(* LS Electric XG5000 project: plc_project_3 *)
(* PLC LSPLC *)

PROGRAM plc_storage (* task: 스캔 프로그램 *)
VAR
    CD : BOOL;
    CV : INT;
    ET : TIME;
    IN1 : BOOL;
    INST : TP;
    INST1 : TON;
    INST10 : TP;
    INST11 : TP;
    INST12 : TP;
    INST13 : TP;
    INST14 : TP;
    INST15 : TP;
    INST16 : TP;
    INST17 : TP;
    INST18 : TP;
    INST19 : TP;
    INST2 : TP;
    INST20 : TP;
    INST21 : TP;
    INST22 : TP;
    INST23 : TP;
    INST24 : TP;
    INST25 : TP;
    INST26 : TP;
    INST27 : TP;
    INST28 : TP;
    INST29 : TP;
    INST3 : TP;
    INST30 : TP;
    INST31 : TP;
    INST32 : TP;
    INST33 : TP;
    INST34 : TP;
    INST35 : TP;
    INST36 : TP;
    INST37 : TP;
    INST4 : TP;
    INST5 : TP;
    INST6 : TP;
    INST7 : TP;
    INST8 : TP;
    INST9 : TP;
    LD : BOOL;
    output1 : INT;
    output2 : UDINT;
    output3 : INT;
    output4 : UDINT;
    output5 : INT;
    output6 : UDINT;
    output7 : INT;
    output8 : UDINT;
    PV : INT;
    QD : BOOL;
    QU : BOOL;
    R : BOOL;
    time1 : TIME;
    time2 : TIME;
    time3 : TIME;
    time4 : TIME;
    난수1 : TON;
    난수2 : TON;
    난수3 : TON;
    놓기 AT %QX0.0.49 : BOOL;
    랜덤수 : INT;
    랜덤수2 : INT;
    반시계 AT %QX0.0.62 : BOOL;
    상 AT %QX0.0.60 : BOOL;
    소요시간1 : TIME;
    소요시간2 : TIME;
    소요시간3 : TIME;
    소요시간4 : TIME;
    소요시간5 : TIME;
    소요시간6 : TIME;
    소요시간7 : TIME;
    소요시간8 : TIME;
    숫자 : INT := 1;
    숫자2 : INT;
    시계 AT %QX0.0.61 : BOOL;
    시퀀스1 AT %MW4 : INT;
    시퀀스2 AT %MW8 : INT;
    앞 AT %QX0.0.59 : BOOL;
    입고 : CTUD_INT;
    입력시간1 AT %MW6 : INT;
    입력시간2 AT %MW2 : INT;
    입력시간3 AT %MW10 : INT;
    입력시간4 AT %MW12 : INT;
    잡기 AT %QX0.0.63 : BOOL;
    저장값 : BOOL;
    출고 : CTUD_INT;
    칸1 AT %QX0.0.50 : BOOL;
    칸10 AT %QX0.0.44 : BOOL;
    칸11 AT %QX0.0.47 : BOOL;
    칸12 AT %QX0.0.46 : BOOL;
    칸2 AT %QX0.0.51 : BOOL;
    칸3 AT %QX0.0.52 : BOOL;
    칸4 AT %QX0.0.53 : BOOL;
    칸5 AT %QX0.0.54 : BOOL;
    칸6 AT %QX0.0.55 : BOOL;
    칸7 AT %QX0.0.56 : BOOL;
    칸8 AT %QX0.0.57 : BOOL;
    칸9 AT %QX0.0.58 : BOOL;
    하 AT %QX0.0.45 : BOOL;
END_VAR
VAR
    _e1 : R_TRIG;
    _p2 : BOOL;
    _e3 : R_TRIG;
    _e4 : R_TRIG;
    _e5 : R_TRIG;
    _t6 : BOOL;
    _e7 : F_TRIG;
    _e8 : F_TRIG;
    _e9 : F_TRIG;
    _e10 : F_TRIG;
    _e11 : F_TRIG;
    _e12 : F_TRIG;
    _e13 : F_TRIG;
    _e14 : F_TRIG;
    _e15 : F_TRIG;
    _e16 : F_TRIG;
    _e17 : F_TRIG;
    _e18 : F_TRIG;
    _e19 : F_TRIG;
    _e20 : F_TRIG;
    _e21 : F_TRIG;
    _e22 : F_TRIG;
    _e23 : F_TRIG;
    _e24 : F_TRIG;
    _e25 : F_TRIG;
    _e26 : F_TRIG;
    _e27 : F_TRIG;
    _e28 : F_TRIG;
    _e29 : F_TRIG;
    _e30 : F_TRIG;
    _e31 : F_TRIG;
    _e32 : F_TRIG;
    _e33 : F_TRIG;
    _e34 : F_TRIG;
    _e35 : F_TRIG;
    _e36 : F_TRIG;
    _e37 : F_TRIG;
    _e38 : F_TRIG;
    _e39 : F_TRIG;
    _e40 : F_TRIG;
    _e41 : F_TRIG;
    _e42 : F_TRIG;
    _e43 : F_TRIG;
    _e44 : F_TRIG;
    _e45 : F_TRIG;
END_VAR

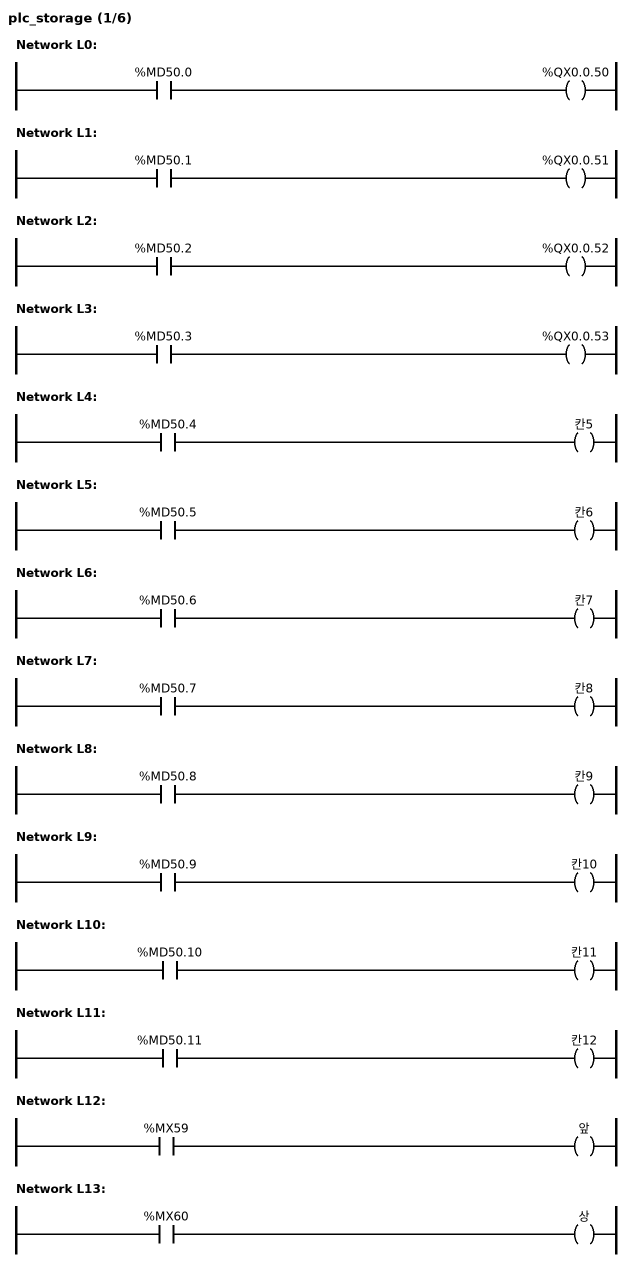
(* Rung L0 *)
%QX0.0.50 := %MD50.0;
(* Rung L1 *)
%QX0.0.51 := %MD50.1;
(* Rung L2 *)
%QX0.0.52 := %MD50.2;
(* Rung L3 *)
%QX0.0.53 := %MD50.3;
(* Rung L4 *)
칸5 := %MD50.4;
(* Rung L5 *)
칸6 := %MD50.5;
(* Rung L6 *)
칸7 := %MD50.6;
(* Rung L7 *)
칸8 := %MD50.7;
(* Rung L8 *)
칸9 := %MD50.8;
(* Rung L9 *)
칸10 := %MD50.9;
(* Rung L10 *)
칸11 := %MD50.10;
(* Rung L11 *)
칸12 := %MD50.11;
(* Rung L12 *)
앞 := %MX59;
(* Rung L13 *)
상 := %MX60;

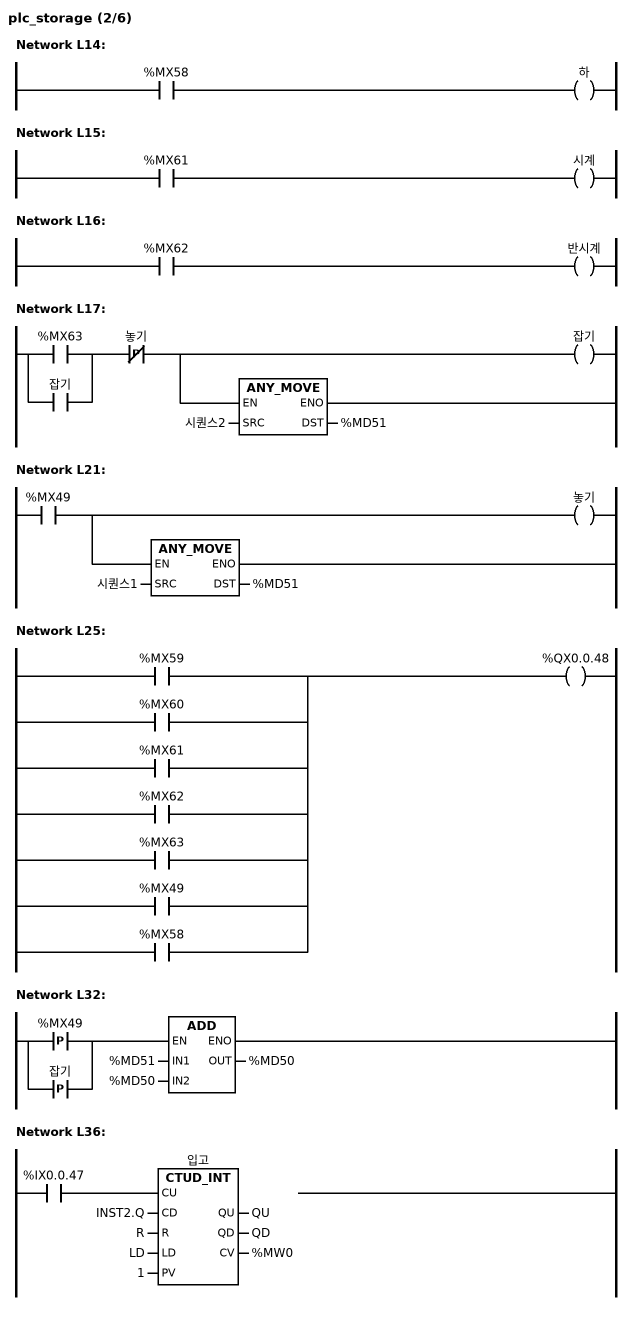
(* Rung L14 *)
하 := %MX58;
(* Rung L15 *)
시계 := %MX61;
(* Rung L16 *)
반시계 := %MX62;
(* Rung L17 *)
_e1(CLK := 놓기);
_p2 := (%MX63 OR 잡기) AND NOT _e1.Q;
잡기 := _p2;
IF _p2 THEN %MD51 := ANY_MOVE(SRC := 시퀀스2); END_IF;
(* Rung L21 *)
놓기 := %MX49;
IF %MX49 THEN %MD51 := ANY_MOVE(SRC := 시퀀스1); END_IF;
(* Rung L25 *)
%QX0.0.48 := %MX59 OR %MX60 OR %MX61 OR %MX62 OR %MX63 OR %MX49 OR %MX58;
(* Rung L32 *)
_e3(CLK := %MX49);
_e4(CLK := 잡기);
IF _e3.Q OR _e4.Q THEN %MD50 := %MD51 + %MD50; END_IF;
(* Rung L36 *)
입고(CU := %IX0.0.47, CD := INST2.Q, R := R, LD := LD, PV := 1, QU => QU, QD => QD, CV => %MW0);

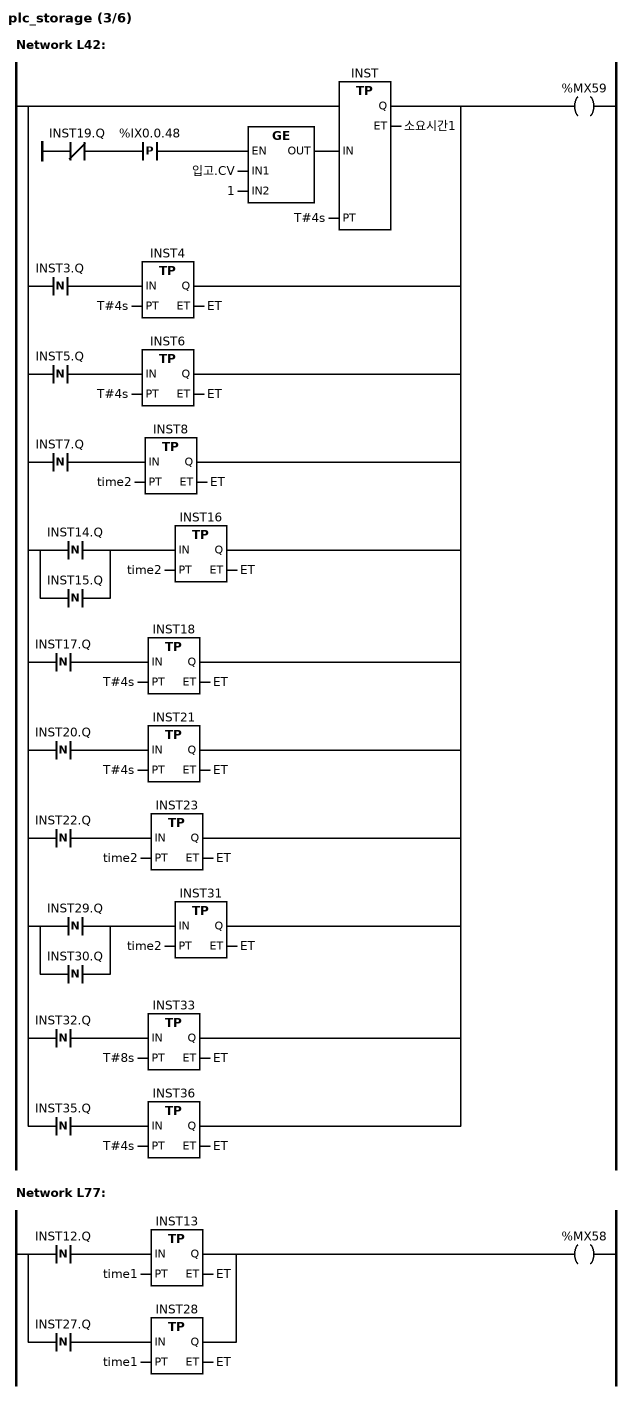
(* Rung L42 *)
_e5(CLK := %IX0.0.48);
IF NOT INST19.Q AND _e5.Q THEN _t6 := 입고.CV >= 1; END_IF;
INST(IN := _t6, PT := T#4s, ET => 소요시간1);
_e7(CLK := INST3.Q);
INST4(IN := _e7.Q, PT := T#4s, ET => ET);
_e8(CLK := INST5.Q);
INST6(IN := _e8.Q, PT := T#4s, ET => ET);
_e9(CLK := INST7.Q);
INST8(IN := _e9.Q, PT := time2, ET => ET);
_e10(CLK := INST14.Q);
_e11(CLK := INST15.Q);
INST16(IN := _e10.Q OR _e11.Q, PT := time2, ET => ET);
_e12(CLK := INST17.Q);
INST18(IN := _e12.Q, PT := T#4s, ET => ET);
_e13(CLK := INST20.Q);
INST21(IN := _e13.Q, PT := T#4s, ET => ET);
_e14(CLK := INST22.Q);
INST23(IN := _e14.Q, PT := time2, ET => ET);
_e15(CLK := INST29.Q);
_e16(CLK := INST30.Q);
INST31(IN := _e15.Q OR _e16.Q, PT := time2, ET => ET);
_e17(CLK := INST32.Q);
INST33(IN := _e17.Q, PT := T#8s, ET => ET);
_e18(CLK := INST35.Q);
INST36(IN := _e18.Q, PT := T#4s, ET => ET);
%MX59 := INST.Q OR INST4.Q OR INST6.Q OR INST8.Q OR INST16.Q OR INST18.Q OR INST21.Q OR INST23.Q OR INST31.Q OR INST33.Q OR INST36.Q;
(* Rung L77 *)
_e19(CLK := INST12.Q);
INST13(IN := _e19.Q, PT := time1, ET => ET);
_e20(CLK := INST27.Q);
INST28(IN := _e20.Q, PT := time1, ET => ET);
%MX58 := INST13.Q OR INST28.Q;

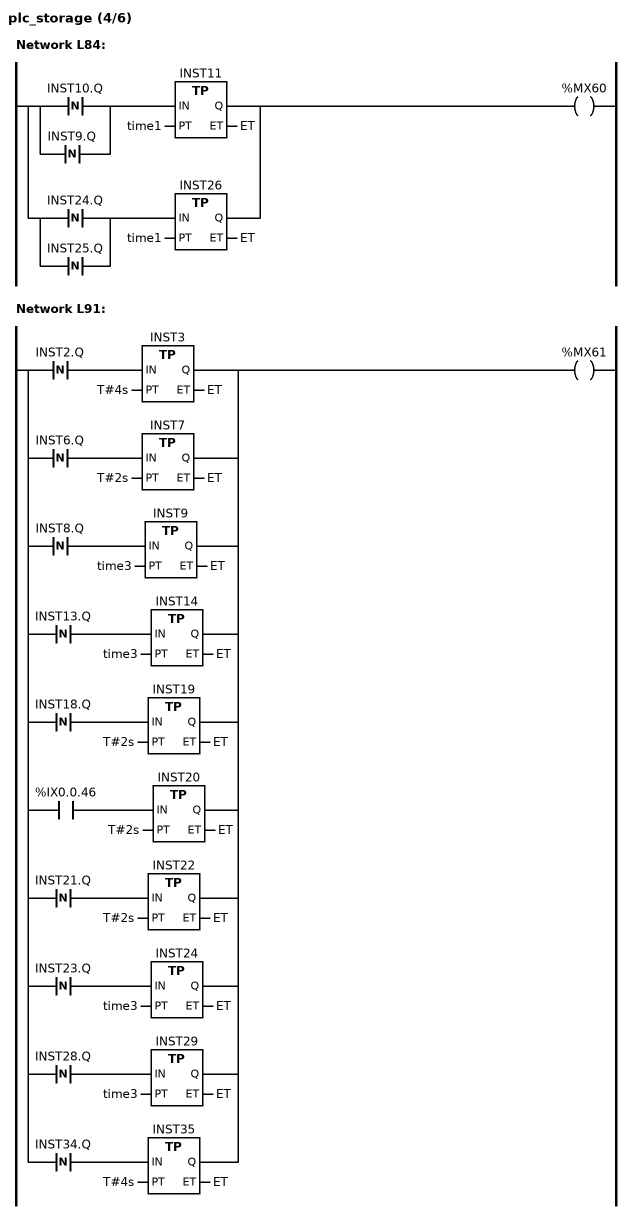
(* Rung L84 *)
_e21(CLK := INST10.Q);
_e22(CLK := INST9.Q);
INST11(IN := _e21.Q OR _e22.Q, PT := time1, ET => ET);
_e23(CLK := INST24.Q);
_e24(CLK := INST25.Q);
INST26(IN := _e23.Q OR _e24.Q, PT := time1, ET => ET);
%MX60 := INST11.Q OR INST26.Q;
(* Rung L91 *)
_e25(CLK := INST2.Q);
INST3(IN := _e25.Q, PT := T#4s, ET => ET);
_e26(CLK := INST6.Q);
INST7(IN := _e26.Q, PT := T#2s, ET => ET);
_e27(CLK := INST8.Q);
INST9(IN := _e27.Q, PT := time3, ET => ET);
_e28(CLK := INST13.Q);
INST14(IN := _e28.Q, PT := time3, ET => ET);
_e29(CLK := INST18.Q);
INST19(IN := _e29.Q, PT := T#2s, ET => ET);
INST20(IN := %IX0.0.46, PT := T#2s, ET => ET);
_e30(CLK := INST21.Q);
INST22(IN := _e30.Q, PT := T#2s, ET => ET);
_e31(CLK := INST23.Q);
INST24(IN := _e31.Q, PT := time3, ET => ET);
_e32(CLK := INST28.Q);
INST29(IN := _e32.Q, PT := time3, ET => ET);
_e33(CLK := INST34.Q);
INST35(IN := _e33.Q, PT := T#4s, ET => ET);
%MX61 := INST3.Q OR INST7.Q OR INST9.Q OR INST14.Q OR INST19.Q OR INST20.Q OR INST22.Q OR INST24.Q OR INST29.Q OR INST35.Q;

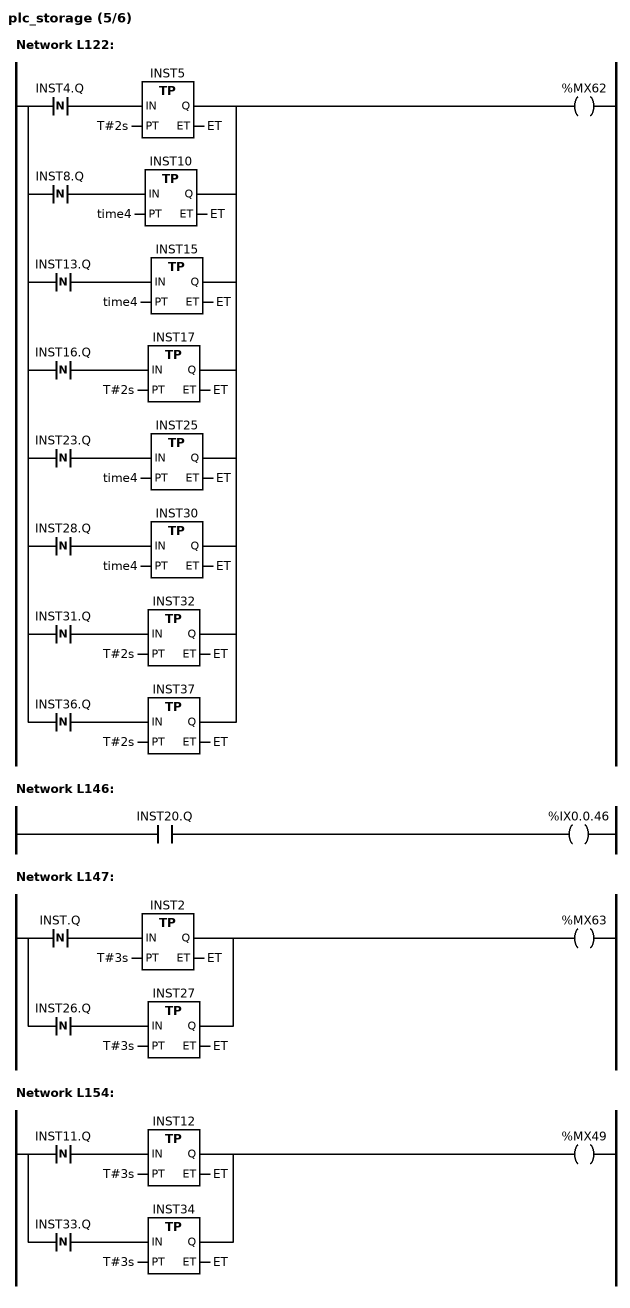
(* Rung L122 *)
_e34(CLK := INST4.Q);
INST5(IN := _e34.Q, PT := T#2s, ET => ET);
_e35(CLK := INST8.Q);
INST10(IN := _e35.Q, PT := time4, ET => ET);
_e36(CLK := INST13.Q);
INST15(IN := _e36.Q, PT := time4, ET => ET);
_e37(CLK := INST16.Q);
INST17(IN := _e37.Q, PT := T#2s, ET => ET);
_e38(CLK := INST23.Q);
INST25(IN := _e38.Q, PT := time4, ET => ET);
_e39(CLK := INST28.Q);
INST30(IN := _e39.Q, PT := time4, ET => ET);
_e40(CLK := INST31.Q);
INST32(IN := _e40.Q, PT := T#2s, ET => ET);
_e41(CLK := INST36.Q);
INST37(IN := _e41.Q, PT := T#2s, ET => ET);
%MX62 := INST5.Q OR INST10.Q OR INST15.Q OR INST17.Q OR INST25.Q OR INST30.Q OR INST32.Q OR INST37.Q;
(* Rung L146 *)
%IX0.0.46 := INST20.Q;
(* Rung L147 *)
_e42(CLK := INST.Q);
INST2(IN := _e42.Q, PT := T#3s, ET => ET);
_e43(CLK := INST26.Q);
INST27(IN := _e43.Q, PT := T#3s, ET => ET);
%MX63 := INST2.Q OR INST27.Q;
(* Rung L154 *)
_e44(CLK := INST11.Q);
INST12(IN := _e44.Q, PT := T#3s, ET => ET);
_e45(CLK := INST33.Q);
INST34(IN := _e45.Q, PT := T#3s, ET => ET);
%MX49 := INST12.Q OR INST34.Q;

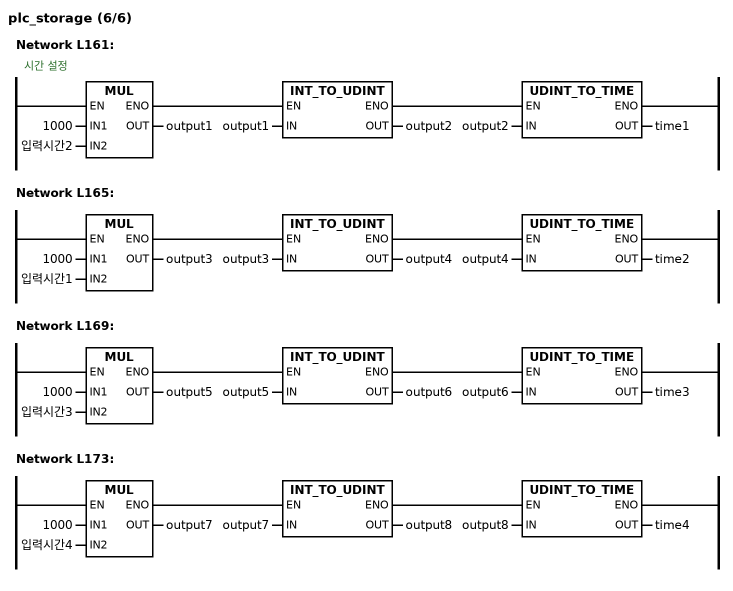
(* 시간 설정 *)
(* Rung L161 *)
output1 := 1000 * 입력시간2;
output2 := INT_TO_UDINT(output1);
time1 := UDINT_TO_TIME(output2);
(* Rung L165 *)
output3 := 1000 * 입력시간1;
output4 := INT_TO_UDINT(output3);
time2 := UDINT_TO_TIME(output4);
(* Rung L169 *)
output5 := 1000 * 입력시간3;
output6 := INT_TO_UDINT(output5);
time3 := UDINT_TO_TIME(output6);
(* Rung L173 *)
output7 := 1000 * 입력시간4;
output8 := INT_TO_UDINT(output7);
time4 := UDINT_TO_TIME(output8);
END_PROGRAM